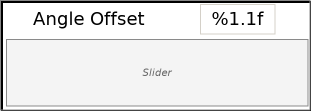
VISUALIZATION InputNumSlider_Angle  // 311x111
VAR_IN_OUT
number : REAL;
END_VAR
    Rectangle (1,1 310x110)
    Slider (6,39 302x67), variable: number, scale 0..360
    Textfield (30,4 150x30), "Angle Offset"
    Textfield (200,4 75x30), "%1.1f", text variable: number
        OnMouseClick: write the text variable via Default, min 0, max 360
END_VISUALIZATION

(* stored: Version 1.1.0.1, ProductVersion 3.1.4024.12
   Visu InputNumSlider_Angle: Id {6ba9cce0-e396-42e4-8e03-de7182a72f48} *)
